// TIA Portal V17 export
// export: Created 2022-07-20T06:59:48.2951314Z, ExportSetting WithDefaults, DisplayName Totally Integrated Automation Portal, DisplayVersion V17, DisplayName TIA Portal Openness, DisplayVersion V17, DisplayName TIA Portal Version Control Interface, DisplayVersion V17, DisplayName SINAMICS Startdrive Advanced, DisplayVersion V17, DisplayName SINAMICS Startdrive G130, G150, S120, S150, SINAMICS MV, S210, DisplayVersion V17, DisplayName SINAMICS Startdrive G110M, G120, G120C, G120D, G120P, G115D, DisplayVersion V17, DisplayName STEP 7 Professional, DisplayVersion V17, DisplayName STEP 7 Safety, DisplayVersion V17, DisplayName WinCC Advanced, DisplayVersion V17
FUNCTION_BLOCK "FB10192_SheetCounter"   // FB10192, LAD
{ S7_Optimized_Access := 'TRUE' }
VERSION : 0.1
// stored: AutoNumber false, IsIECCheckEnabled false, IsRetainMemResEnabled false, MemoryReserve 100, SetENOAutomatically false, UDAEnableTagReadback false
   VAR_INPUT
      FirstSheetSensor : Bool;
   END_VAR
   VAR_OUTPUT
      NumberOfSheetDetected : UInt;
   END_VAR
   VAR
      R_TRIG_NumberOfSheetDetected : R_TRIG;
   END_VAR
BEGIN

REGION Network 1 (SCL): First Scan
   IF "FirstScan" THEN
       #NumberOfSheetDetected := 0;
   END_IF;
END_REGION

REGION Network 2 (SCL): Edge Signals & Timers
   REGION EDGE SIGNAL
       #R_TRIG_NumberOfSheetDetected(CLK := #FirstSheetSensor);
   END_REGION
END_REGION

REGION Network 3 (SCL): Sheets Counter
   IF #R_TRIG_NumberOfSheetDetected.Q THEN
       #NumberOfSheetDetected += 1;
   END_IF;
END_REGION
END_FUNCTION_BLOCK
